FUNCTION_BLOCK FloorIndicator_HMI (* Service Interface Function Block Type *)
  (* Standard: 61499-2 *)
  (* Version 0.0, 6/3/2016, Andrei, nxtControl GmbH, template *)
  PACKAGE Main;
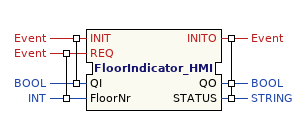
  EVENT_INPUT
    INIT WITH QI;
    REQ WITH FloorNr;
  END_EVENT
  EVENT_OUTPUT
    INITO WITH QO, STATUS;
  END_EVENT
  VAR_INPUT
    QI : BOOL;
    FloorNr : INT;
  END_VAR
  VAR_OUTPUT
    QO : BOOL; (* Event Output Qualifier *)
    STATUS : STRING; (* Service Status *)
  END_VAR
  SERVICE /
    SEQUENCE 
    END_SEQUENCE
  END_SERVICE
END_FUNCTION_BLOCK
